TYPE ST_ActionData :
STRUCT
	eAction		: E_Action;
	nObject		: UINT;
	nTarget		: UINT;
	aParams		: ARRAY[1..19] OF DINT;
END_STRUCT
END_TYPE

(* stored: Version 1.1.0.1, ProductVersion 3.1.4024.9
   DUT ST_ActionData: Id {7ae75ca5-483f-450d-96e8-7dd1d3742df3} *)
